Omron CX-Programmer project 新工程 (CX-Programmer 9.73)

# PLC 新PLC1: CJ1M CPU21

## Program 新程序1 (cyclic task 0)
; 这个PLC程序是我为正佳广场四楼设计的楼宇自动化控制系统。系统控制的物理设备包括照明设备、空调设备和电梯设备。系统启动时，只有在PLC上电信号为真时，照明系统电源、空调系统电源和电梯系统电源才会被激活，确保设备电源正常供应。随后，当系统启动信号为真时，系统进入运行状态，操作人员可以通过触摸屏模式选择信号选择照明模式。此时，照明控制信号置位，照明系统电源启动照明设备，为商场提供适宜的照明环境。若需调整亮度，触摸屏亮度调整信号会触发亮度调节，但这必须在系统启动信号为真的情况下才能生效，以避免未启动时误操作。通过定时器控制设备运行时间，确保设备在规定时间内完成任务。若定时器未能在预设时间内完成，系统故障指示灯会被点亮，提示操作人员检查系统状态。操作人员通过触摸屏操作信号触发系统运行输出，但系统运行输出仅在系统启动信号为真时才会被置位，防止未授权的操作影响系统。通过CMP指令比较数据寄存器的值，若检测到异常，照明故障指示灯或空调故障指示灯会被点亮，具体取决于故障来源。同时，报警灯在任何故障发生时都会点亮，向操作人员发出警示。

### Section 段1

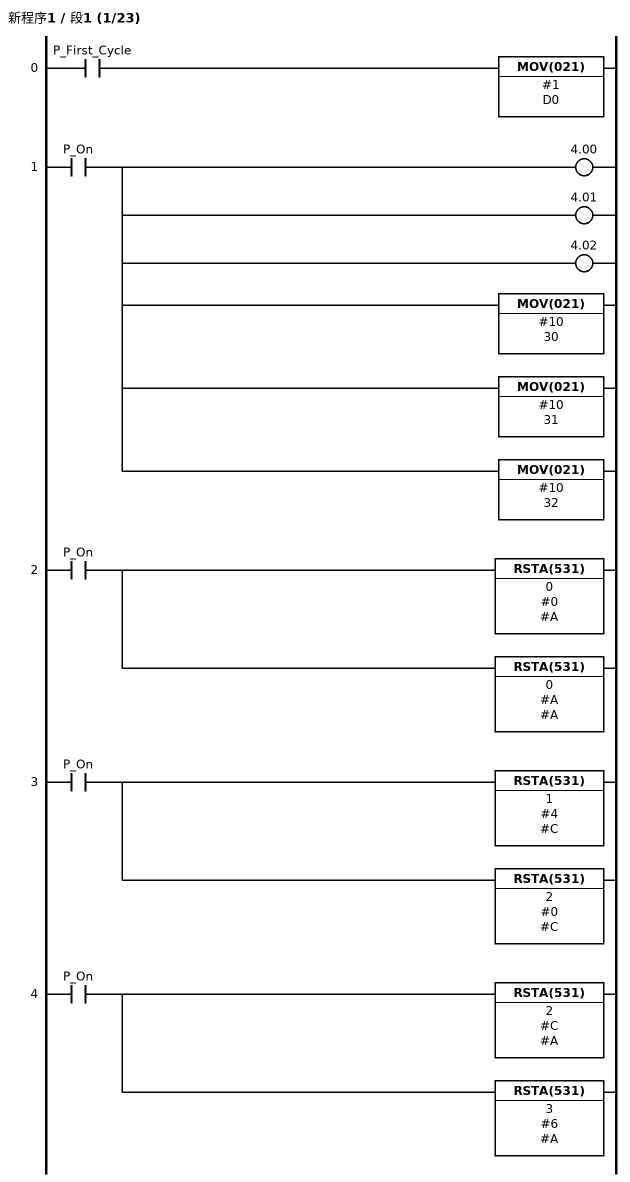
; rung 0
LD P_First_Cycle
MOV(021) #1 D0
; rung 1
LD P_On
OUT 4.00
OUT 4.01
OUT 4.02
MOV(021) #10 30
MOV(021) #10 31
MOV(021) #10 32
; rung 2
LD P_On
RSTA(531) 0 #0 #A
RSTA(531) 0 #A #A
; rung 3
LD P_On
RSTA(531) 1 #4 #C
RSTA(531) 2 #0 #C
; rung 4
LD P_On
RSTA(531) 2 #C #A
RSTA(531) 3 #6 #A

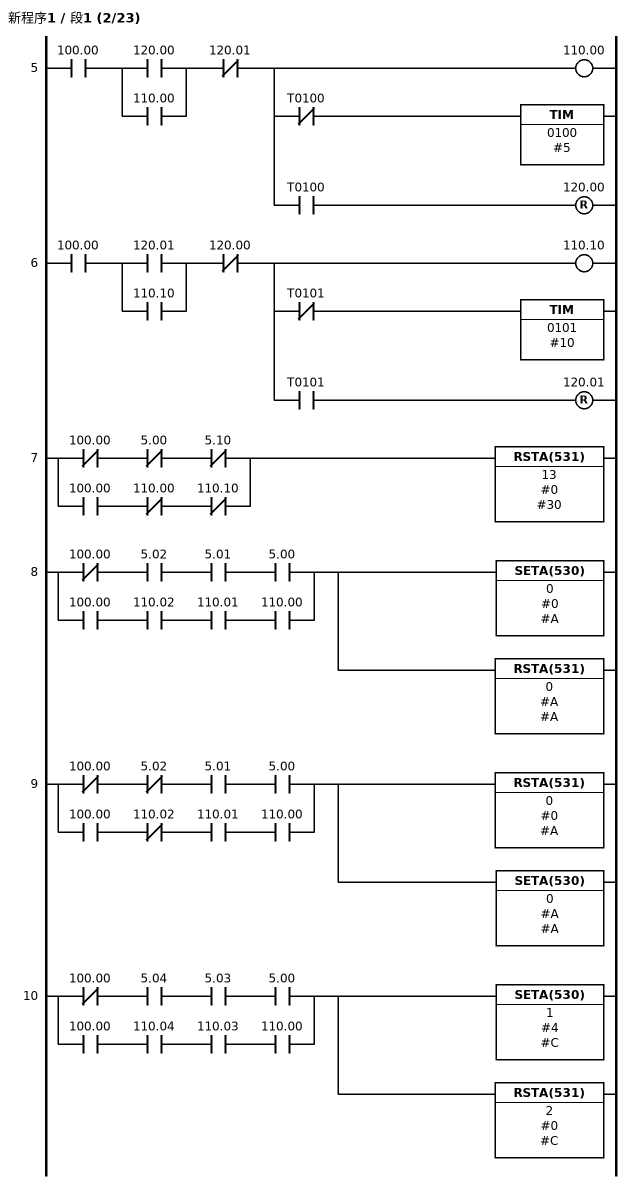
; rung 5
LD 100.00
LD 120.00
OR 110.00
ANDLD
ANDNOT 120.01
OUT TR0
OUT 110.00
ANDNOT T0100
TIM 0100 #5
LD TR0
AND T0100
RSET 120.00
; rung 6
LD 100.00
LD 120.01
OR 110.10
ANDLD
ANDNOT 120.00
OUT TR0
OUT 110.10
ANDNOT T0101
TIM 0101 #10
LD TR0
AND T0101
RSET 120.01
; rung 7
LDNOT 100.00
ANDNOT 5.00
ANDNOT 5.10
LD 100.00
ANDNOT 110.00
ANDNOT 110.10
ORLD
RSTA(531) 13 #0 #30
; rung 8
LDNOT 100.00
AND 5.02
AND 5.01
AND 5.00
LD 100.00
AND 110.02
AND 110.01
AND 110.00
ORLD
SETA(530) 0 #0 #A
RSTA(531) 0 #A #A
; rung 9
LDNOT 100.00
ANDNOT 5.02
AND 5.01
AND 5.00
LD 100.00
ANDNOT 110.02
AND 110.01
AND 110.00
ORLD
RSTA(531) 0 #0 #A
SETA(530) 0 #A #A
; rung 10
LDNOT 100.00
AND 5.04
AND 5.03
AND 5.00
LD 100.00
AND 110.04
AND 110.03
AND 110.00
ORLD
SETA(530) 1 #4 #C
RSTA(531) 2 #0 #C

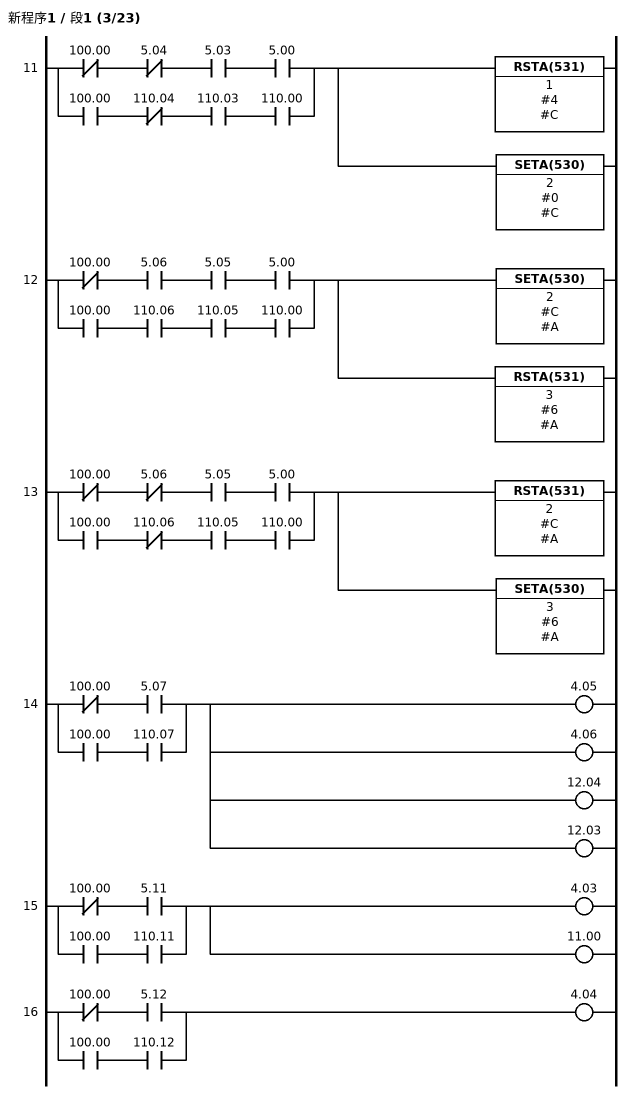
; rung 11
LDNOT 100.00
ANDNOT 5.04
AND 5.03
AND 5.00
LD 100.00
ANDNOT 110.04
AND 110.03
AND 110.00
ORLD
RSTA(531) 1 #4 #C
SETA(530) 2 #0 #C
; rung 12
LDNOT 100.00
AND 5.06
AND 5.05
AND 5.00
LD 100.00
AND 110.06
AND 110.05
AND 110.00
ORLD
SETA(530) 2 #C #A
RSTA(531) 3 #6 #A
; rung 13
LDNOT 100.00
ANDNOT 5.06
AND 5.05
AND 5.00
LD 100.00
ANDNOT 110.06
AND 110.05
AND 110.00
ORLD
RSTA(531) 2 #C #A
SETA(530) 3 #6 #A
; rung 14
LDNOT 100.00
AND 5.07
LD 100.00
AND 110.07
ORLD
OUT 4.05
OUT 4.06
OUT 12.04
OUT 12.03
; rung 15
LDNOT 100.00
AND 5.11
LD 100.00
AND 110.11
ORLD
OUT 4.03
OUT 11.00
; rung 16
LDNOT 100.00
AND 5.12
LD 100.00
AND 110.12
ORLD
OUT 4.04

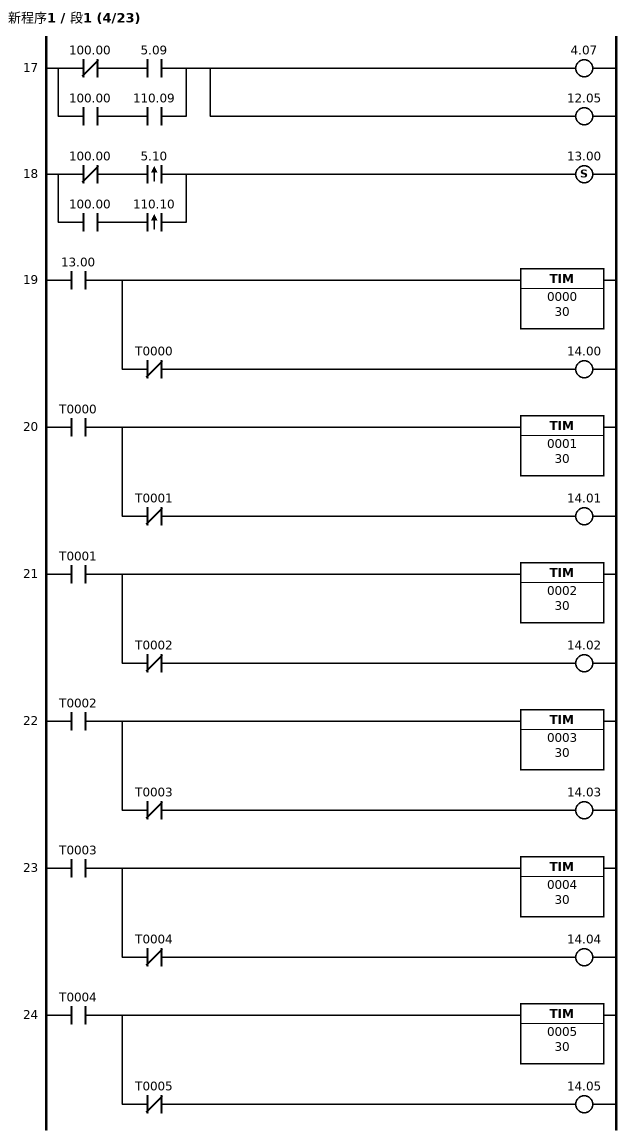
; rung 17
LDNOT 100.00
AND 5.09
LD 100.00
AND 110.09
ORLD
OUT 4.07
OUT 12.05
; rung 18
LDNOT 100.00
@AND 5.10
LD 100.00
@AND 110.10
ORLD
SET 13.00
; rung 19
LD 13.00
TIM 0000 30
ANDNOT T0000
OUT 14.00
; rung 20
LD T0000
TIM 0001 30
ANDNOT T0001
OUT 14.01
; rung 21
LD T0001
TIM 0002 30
ANDNOT T0002
OUT 14.02
; rung 22
LD T0002
TIM 0003 30
ANDNOT T0003
OUT 14.03
; rung 23
LD T0003
TIM 0004 30
ANDNOT T0004
OUT 14.04
; rung 24
LD T0004
TIM 0005 30
ANDNOT T0005
OUT 14.05

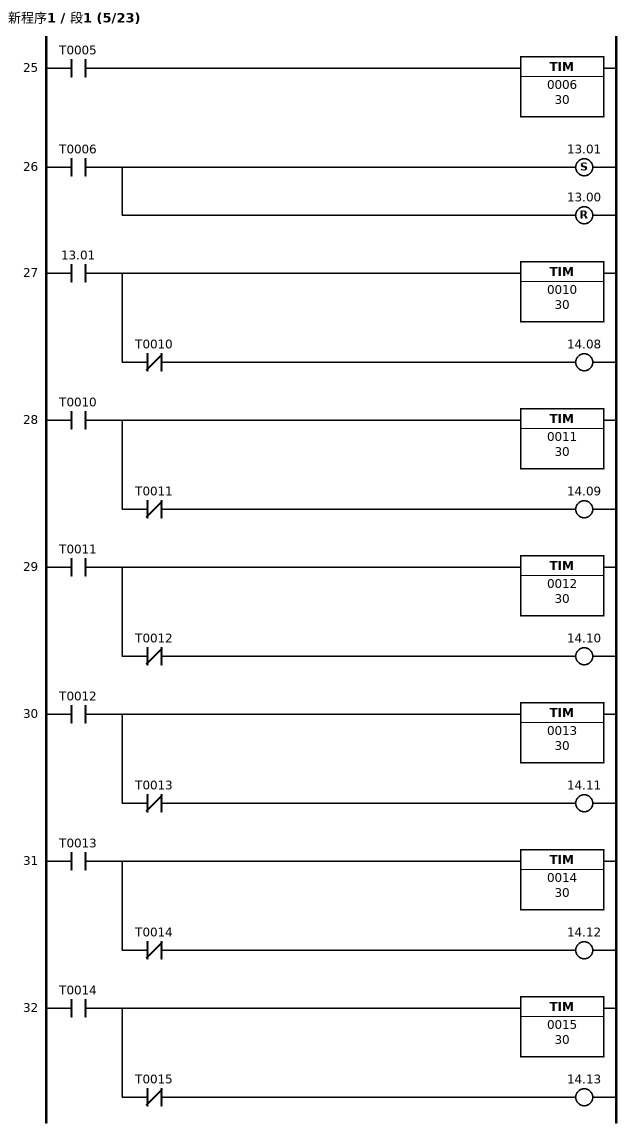
; rung 25
LD T0005
TIM 0006 30
; rung 26
LD T0006
SET 13.01
RSET 13.00
; rung 27
LD 13.01
TIM 0010 30
ANDNOT T0010
OUT 14.08
; rung 28
LD T0010
TIM 0011 30
ANDNOT T0011
OUT 14.09
; rung 29
LD T0011
TIM 0012 30
ANDNOT T0012
OUT 14.10
; rung 30
LD T0012
TIM 0013 30
ANDNOT T0013
OUT 14.11
; rung 31
LD T0013
TIM 0014 30
ANDNOT T0014
OUT 14.12
; rung 32
LD T0014
TIM 0015 30
ANDNOT T0015
OUT 14.13

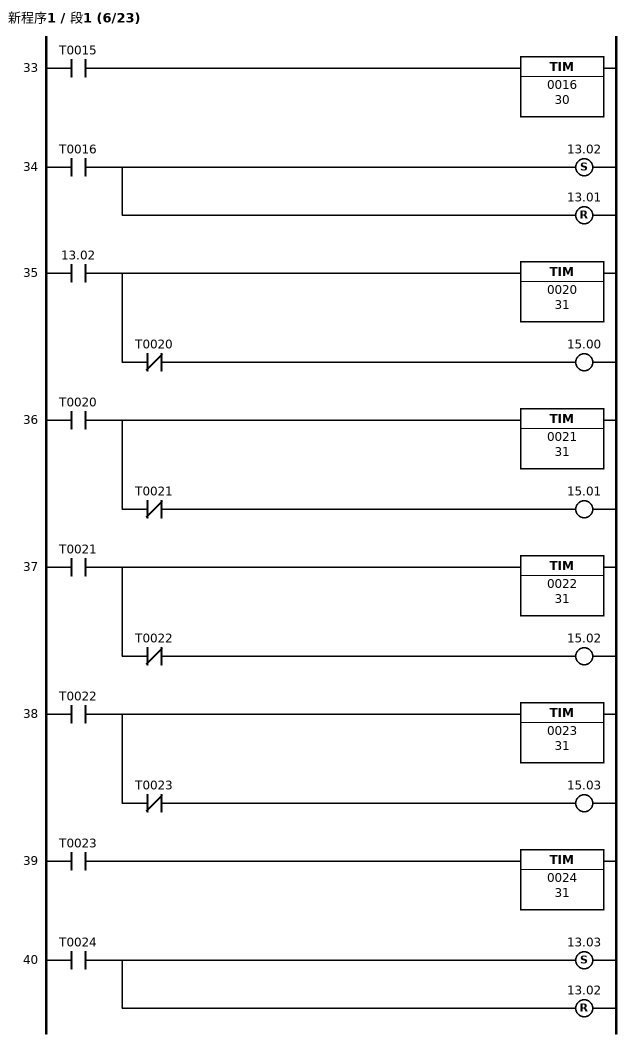
; rung 33
LD T0015
TIM 0016 30
; rung 34
LD T0016
SET 13.02
RSET 13.01
; rung 35
LD 13.02
TIM 0020 31
ANDNOT T0020
OUT 15.00
; rung 36
LD T0020
TIM 0021 31
ANDNOT T0021
OUT 15.01
; rung 37
LD T0021
TIM 0022 31
ANDNOT T0022
OUT 15.02
; rung 38
LD T0022
TIM 0023 31
ANDNOT T0023
OUT 15.03
; rung 39
LD T0023
TIM 0024 31
; rung 40
LD T0024
SET 13.03
RSET 13.02

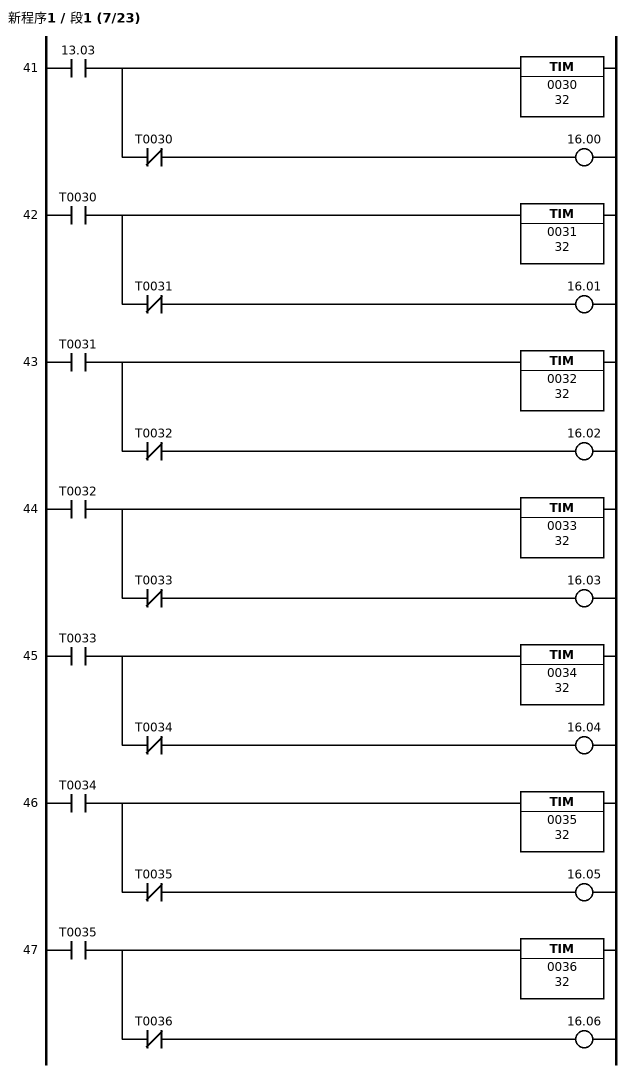
; rung 41
LD 13.03
TIM 0030 32
ANDNOT T0030
OUT 16.00
; rung 42
LD T0030
TIM 0031 32
ANDNOT T0031
OUT 16.01
; rung 43
LD T0031
TIM 0032 32
ANDNOT T0032
OUT 16.02
; rung 44
LD T0032
TIM 0033 32
ANDNOT T0033
OUT 16.03
; rung 45
LD T0033
TIM 0034 32
ANDNOT T0034
OUT 16.04
; rung 46
LD T0034
TIM 0035 32
ANDNOT T0035
OUT 16.05
; rung 47
LD T0035
TIM 0036 32
ANDNOT T0036
OUT 16.06

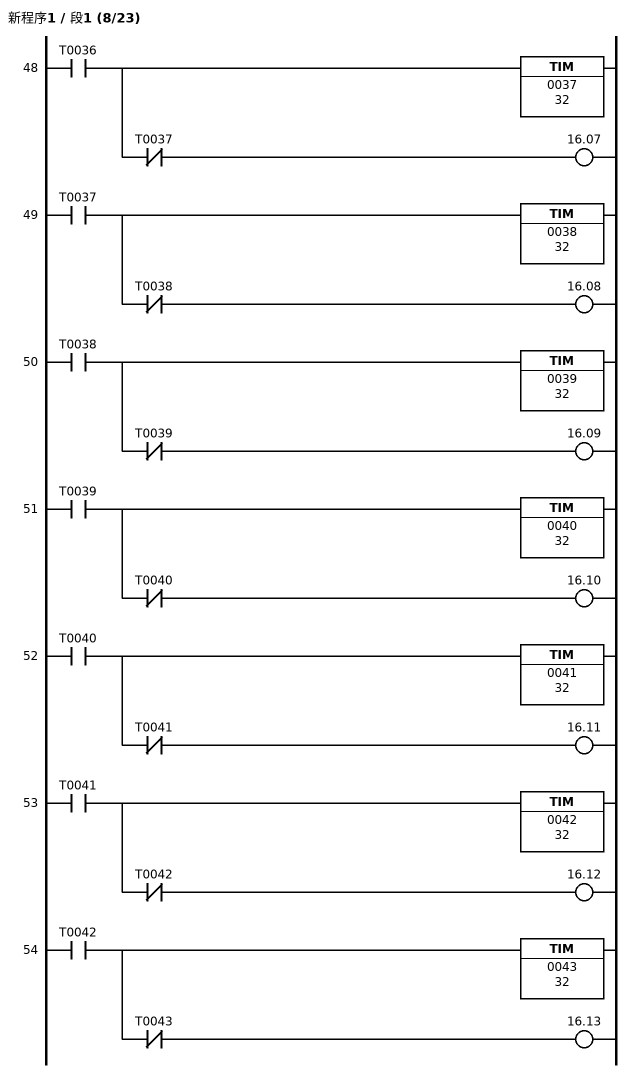
; rung 48
LD T0036
TIM 0037 32
ANDNOT T0037
OUT 16.07
; rung 49
LD T0037
TIM 0038 32
ANDNOT T0038
OUT 16.08
; rung 50
LD T0038
TIM 0039 32
ANDNOT T0039
OUT 16.09
; rung 51
LD T0039
TIM 0040 32
ANDNOT T0040
OUT 16.10
; rung 52
LD T0040
TIM 0041 32
ANDNOT T0041
OUT 16.11
; rung 53
LD T0041
TIM 0042 32
ANDNOT T0042
OUT 16.12
; rung 54
LD T0042
TIM 0043 32
ANDNOT T0043
OUT 16.13

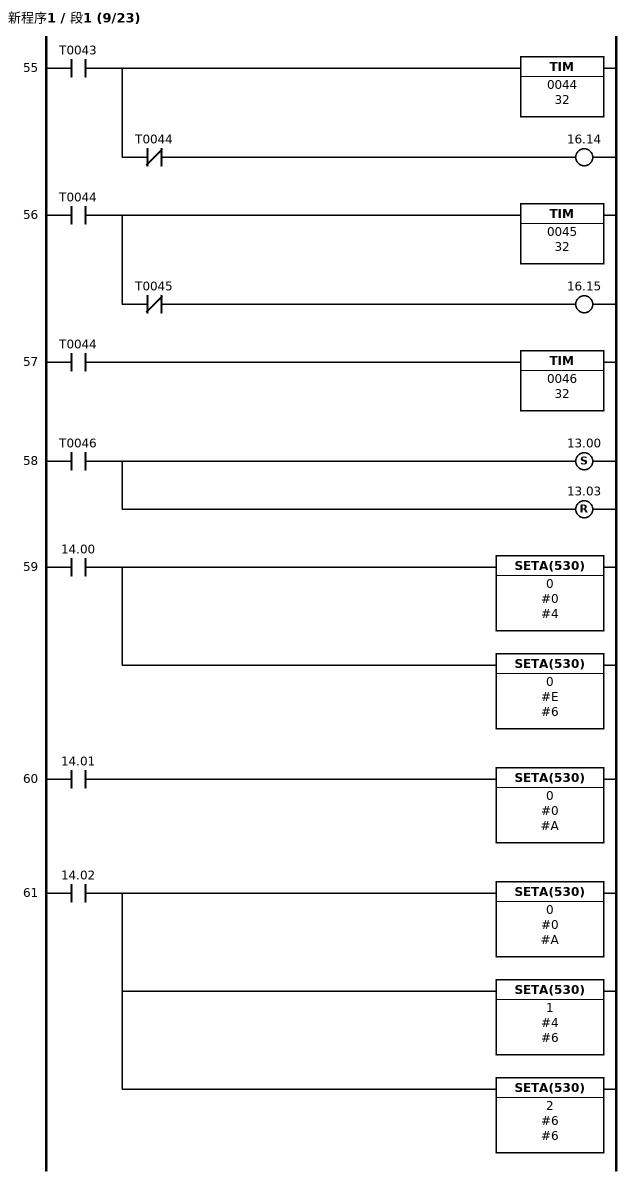
; rung 55
LD T0043
TIM 0044 32
ANDNOT T0044
OUT 16.14
; rung 56
LD T0044
TIM 0045 32
ANDNOT T0045
OUT 16.15
; rung 57
LD T0044
TIM 0046 32
; rung 58
LD T0046
SET 13.00
RSET 13.03
; rung 59
LD 14.00
SETA(530) 0 #0 #4
SETA(530) 0 #E #6
; rung 60
LD 14.01
SETA(530) 0 #0 #A
; rung 61
LD 14.02
SETA(530) 0 #0 #A
SETA(530) 1 #4 #6
SETA(530) 2 #6 #6

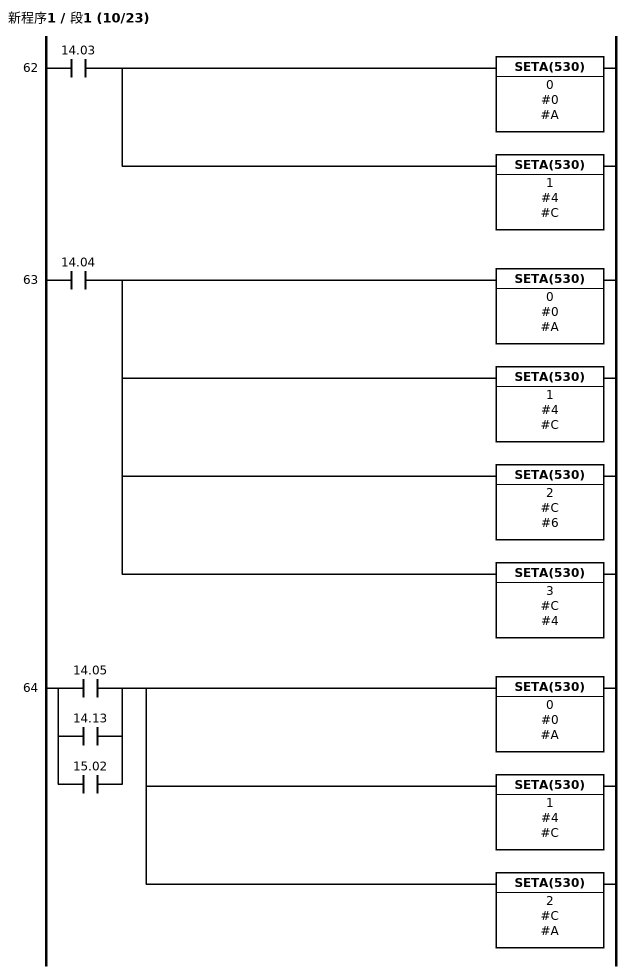
; rung 62
LD 14.03
SETA(530) 0 #0 #A
SETA(530) 1 #4 #C
; rung 63
LD 14.04
SETA(530) 0 #0 #A
SETA(530) 1 #4 #C
SETA(530) 2 #C #6
SETA(530) 3 #C #4
; rung 64
LD 14.05
OR 14.13
OR 15.02
SETA(530) 0 #0 #A
SETA(530) 1 #4 #C
SETA(530) 2 #C #A

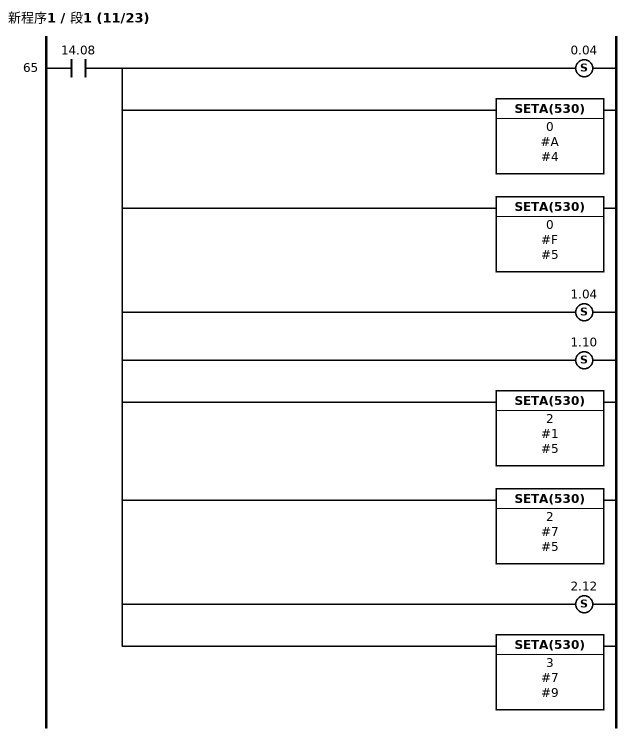
; rung 65
LD 14.08
SET 0.04
SETA(530) 0 #A #4
SETA(530) 0 #F #5
SET 1.04
SET 1.10
SETA(530) 2 #1 #5
SETA(530) 2 #7 #5
SET 2.12
SETA(530) 3 #7 #9

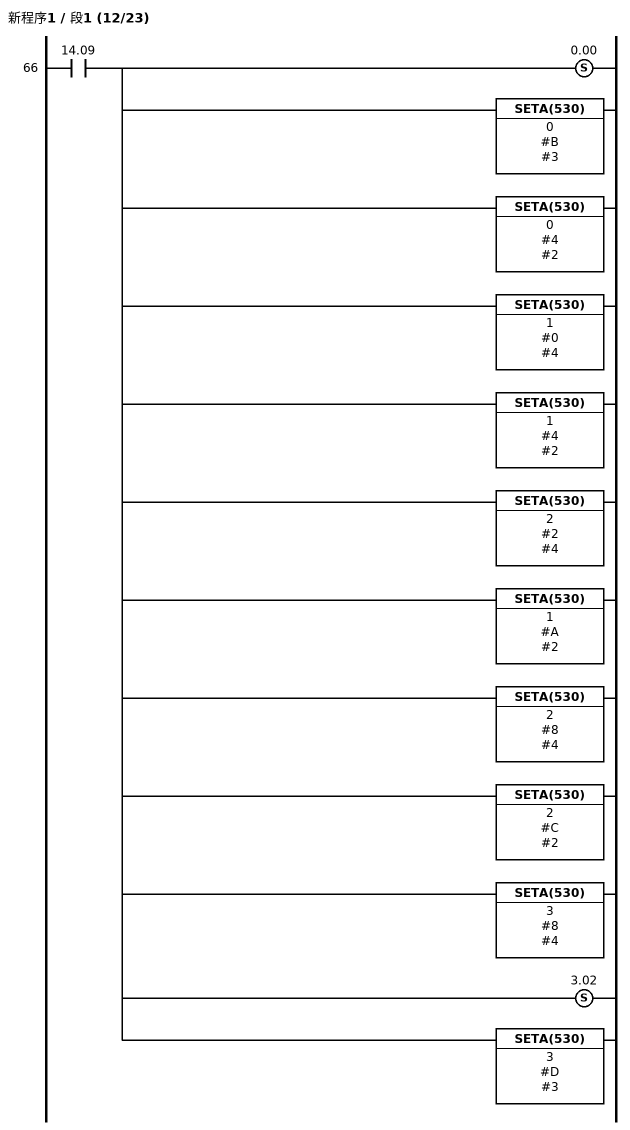
; rung 66
LD 14.09
SET 0.00
SETA(530) 0 #B #3
SETA(530) 0 #4 #2
SETA(530) 1 #0 #4
SETA(530) 1 #4 #2
SETA(530) 2 #2 #4
SETA(530) 1 #A #2
SETA(530) 2 #8 #4
SETA(530) 2 #C #2
SETA(530) 3 #8 #4
SET 3.02
SETA(530) 3 #D #3

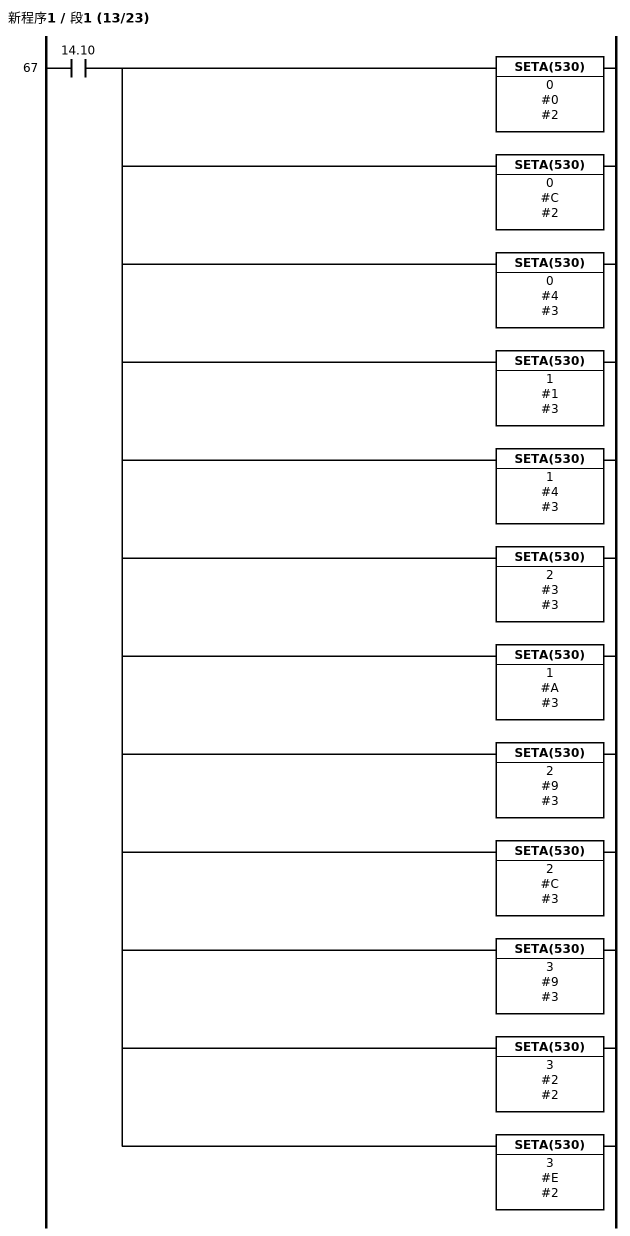
; rung 67
LD 14.10
SETA(530) 0 #0 #2
SETA(530) 0 #C #2
SETA(530) 0 #4 #3
SETA(530) 1 #1 #3
SETA(530) 1 #4 #3
SETA(530) 2 #3 #3
SETA(530) 1 #A #3
SETA(530) 2 #9 #3
SETA(530) 2 #C #3
SETA(530) 3 #9 #3
SETA(530) 3 #2 #2
SETA(530) 3 #E #2

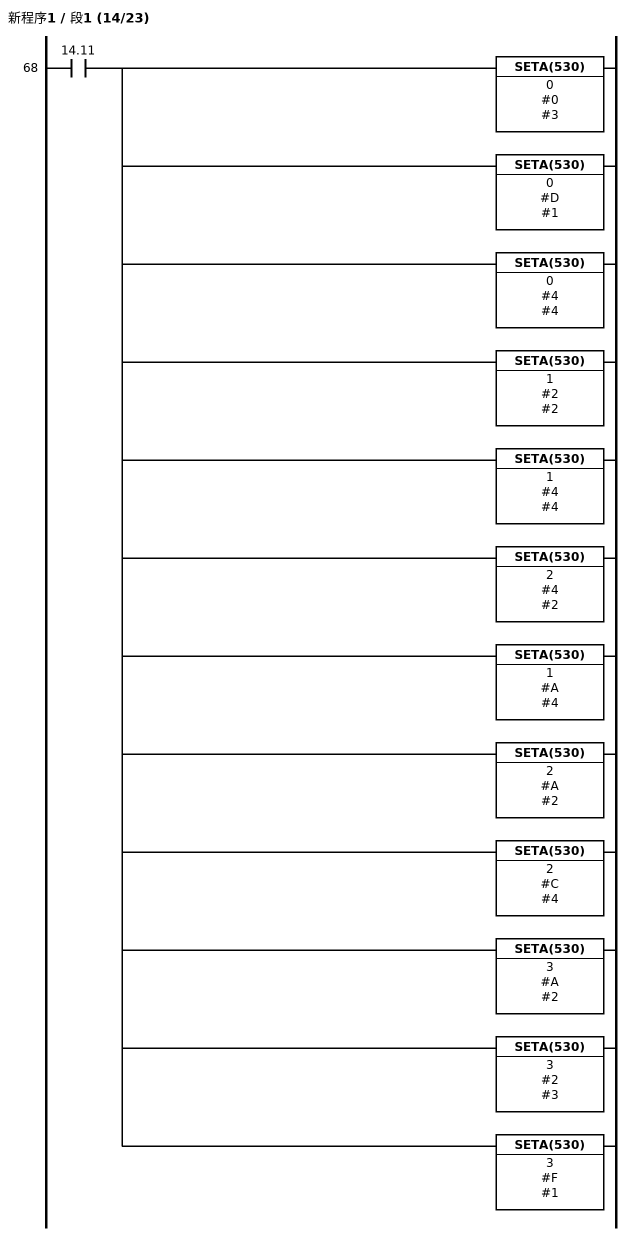
; rung 68
LD 14.11
SETA(530) 0 #0 #3
SETA(530) 0 #D #1
SETA(530) 0 #4 #4
SETA(530) 1 #2 #2
SETA(530) 1 #4 #4
SETA(530) 2 #4 #2
SETA(530) 1 #A #4
SETA(530) 2 #A #2
SETA(530) 2 #C #4
SETA(530) 3 #A #2
SETA(530) 3 #2 #3
SETA(530) 3 #F #1

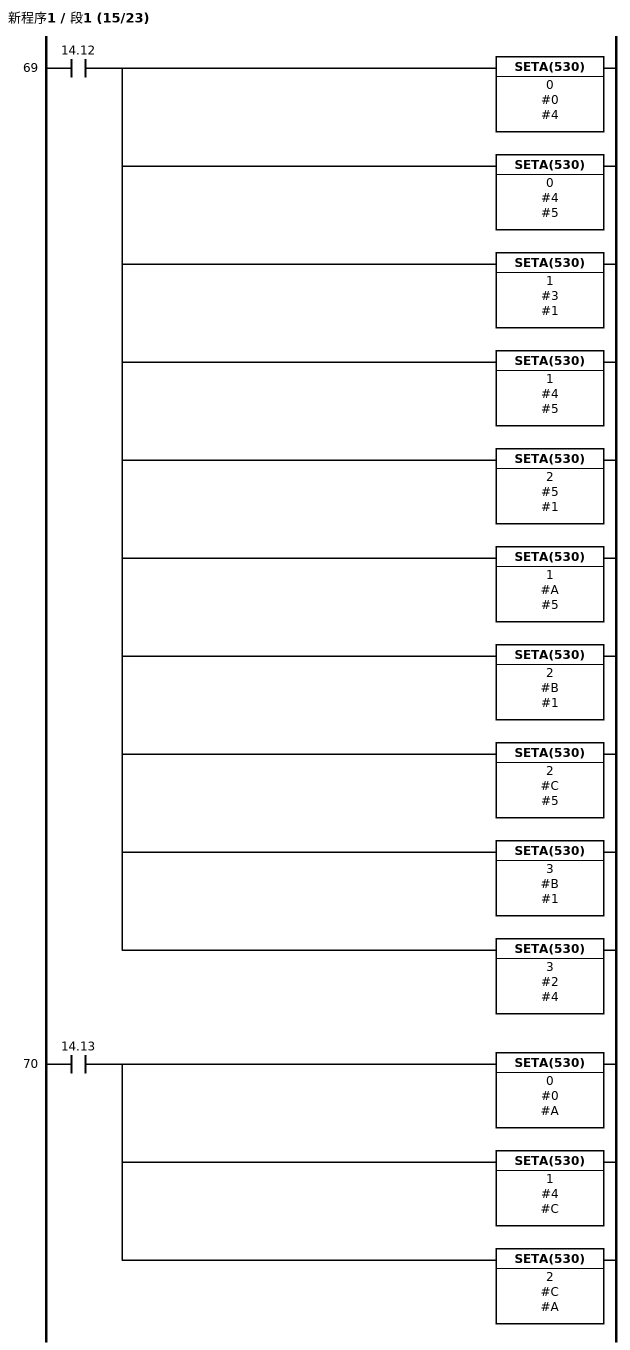
; rung 69
LD 14.12
SETA(530) 0 #0 #4
SETA(530) 0 #4 #5
SETA(530) 1 #3 #1
SETA(530) 1 #4 #5
SETA(530) 2 #5 #1
SETA(530) 1 #A #5
SETA(530) 2 #B #1
SETA(530) 2 #C #5
SETA(530) 3 #B #1
SETA(530) 3 #2 #4
; rung 70
LD 14.13
SETA(530) 0 #0 #A
SETA(530) 1 #4 #C
SETA(530) 2 #C #A

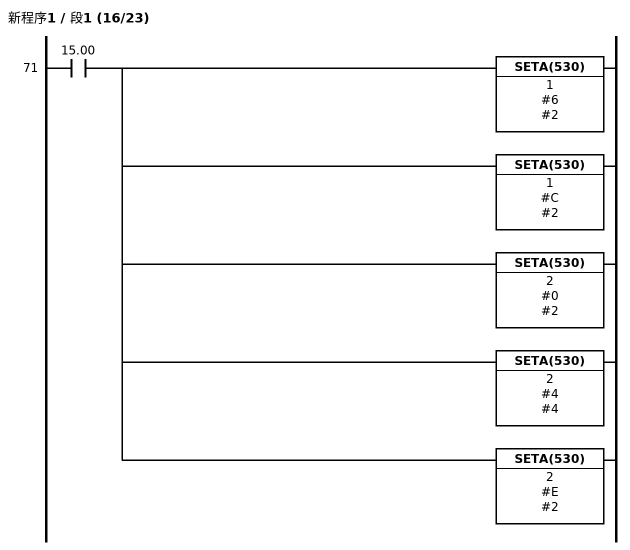
; rung 71
LD 15.00
SETA(530) 1 #6 #2
SETA(530) 1 #C #2
SETA(530) 2 #0 #2
SETA(530) 2 #4 #4
SETA(530) 2 #E #2

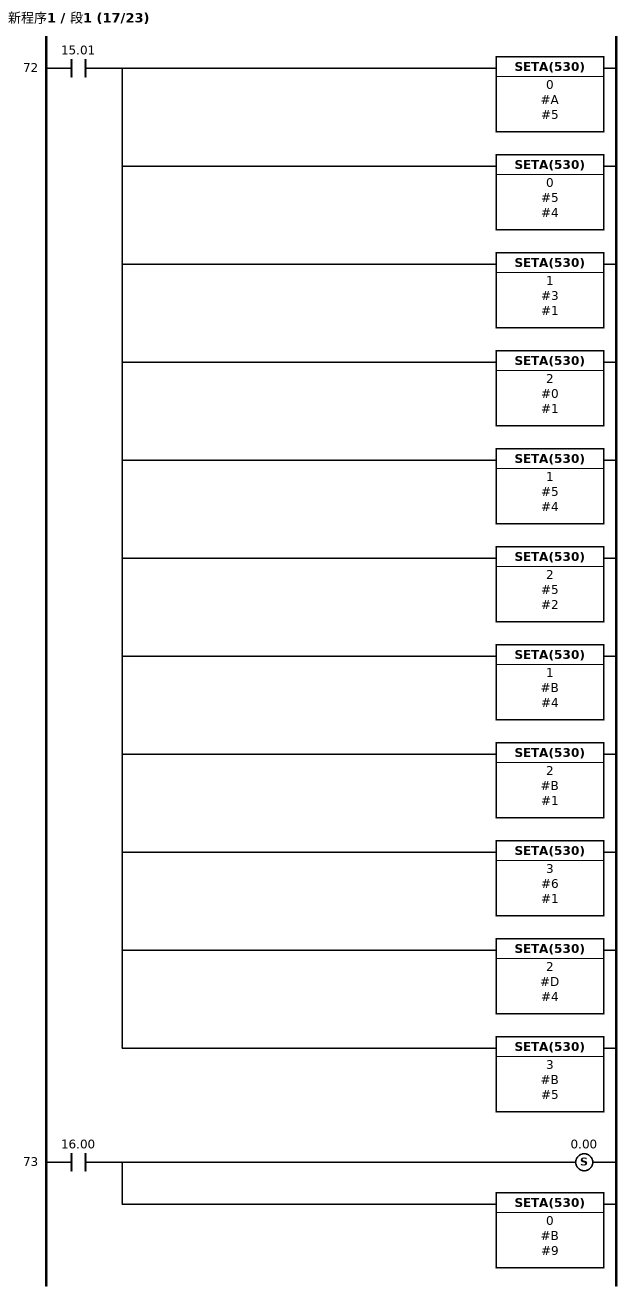
; rung 72
LD 15.01
SETA(530) 0 #A #5
SETA(530) 0 #5 #4
SETA(530) 1 #3 #1
SETA(530) 2 #0 #1
SETA(530) 1 #5 #4
SETA(530) 2 #5 #2
SETA(530) 1 #B #4
SETA(530) 2 #B #1
SETA(530) 3 #6 #1
SETA(530) 2 #D #4
SETA(530) 3 #B #5
; rung 73
LD 16.00
SET 0.00
SETA(530) 0 #B #9

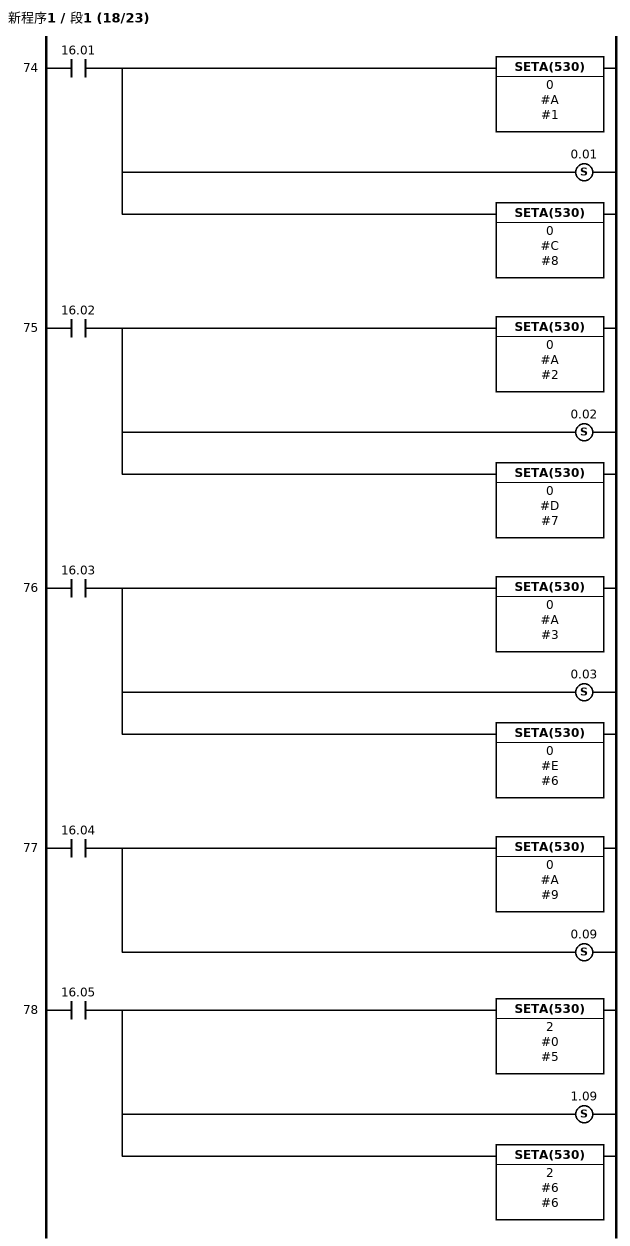
; rung 74
LD 16.01
SETA(530) 0 #A #1
SET 0.01
SETA(530) 0 #C #8
; rung 75
LD 16.02
SETA(530) 0 #A #2
SET 0.02
SETA(530) 0 #D #7
; rung 76
LD 16.03
SETA(530) 0 #A #3
SET 0.03
SETA(530) 0 #E #6
; rung 77
LD 16.04
SETA(530) 0 #A #9
SET 0.09
; rung 78
LD 16.05
SETA(530) 2 #0 #5
SET 1.09
SETA(530) 2 #6 #6

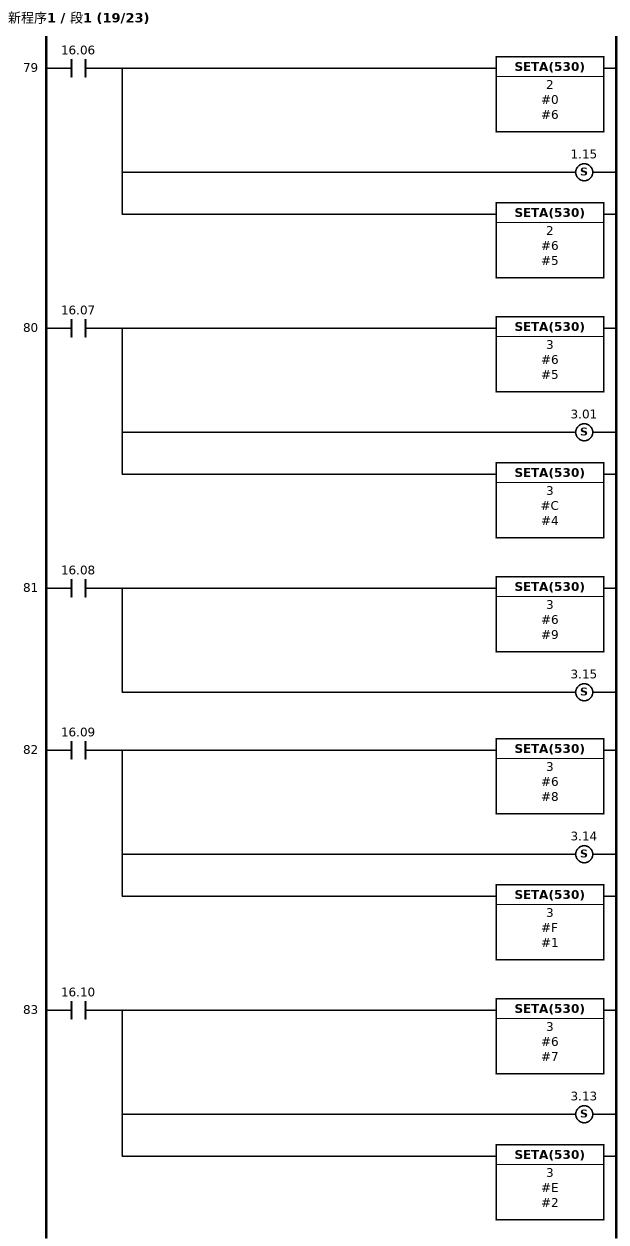
; rung 79
LD 16.06
SETA(530) 2 #0 #6
SET 1.15
SETA(530) 2 #6 #5
; rung 80
LD 16.07
SETA(530) 3 #6 #5
SET 3.01
SETA(530) 3 #C #4
; rung 81
LD 16.08
SETA(530) 3 #6 #9
SET 3.15
; rung 82
LD 16.09
SETA(530) 3 #6 #8
SET 3.14
SETA(530) 3 #F #1
; rung 83
LD 16.10
SETA(530) 3 #6 #7
SET 3.13
SETA(530) 3 #E #2

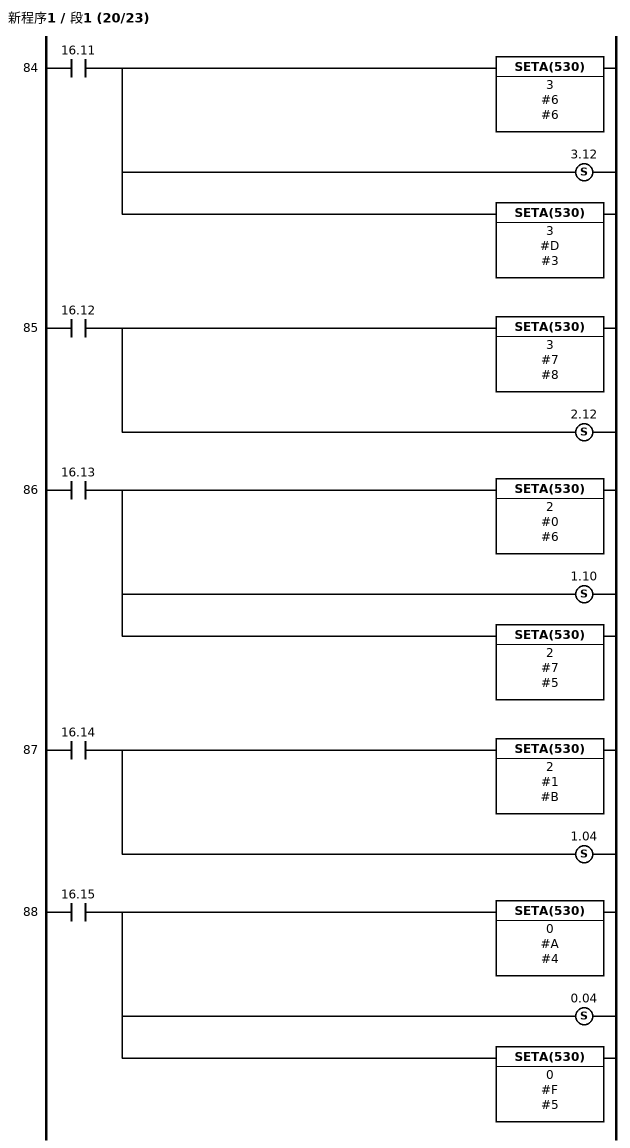
; rung 84
LD 16.11
SETA(530) 3 #6 #6
SET 3.12
SETA(530) 3 #D #3
; rung 85
LD 16.12
SETA(530) 3 #7 #8
SET 2.12
; rung 86
LD 16.13
SETA(530) 2 #0 #6
SET 1.10
SETA(530) 2 #7 #5
; rung 87
LD 16.14
SETA(530) 2 #1 #B
SET 1.04
; rung 88
LD 16.15
SETA(530) 0 #A #4
SET 0.04
SETA(530) 0 #F #5

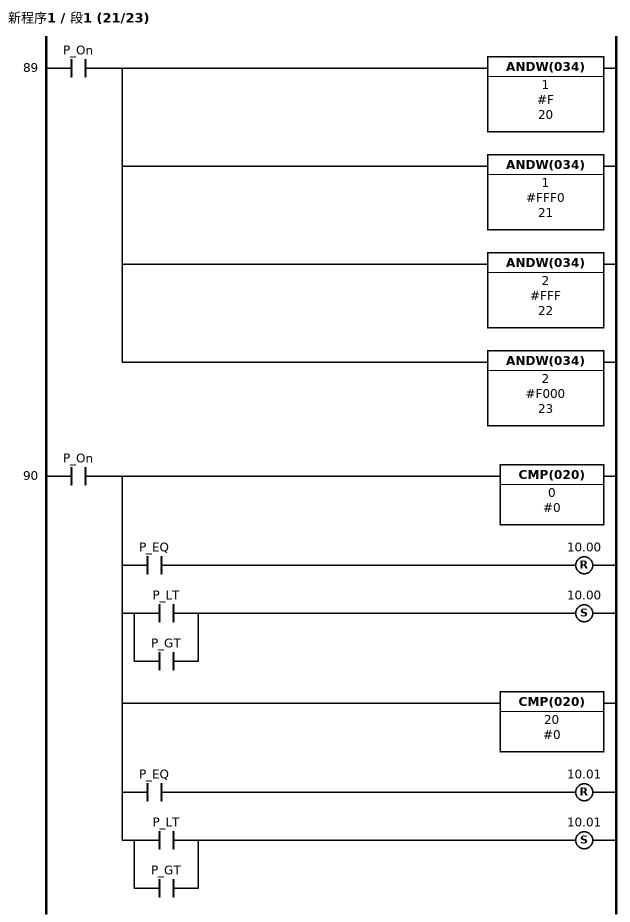
; rung 89
LD P_On
ANDW(034) 1 #F 20
ANDW(034) 1 #FFF0 21
ANDW(034) 2 #FFF 22
ANDW(034) 2 #F000 23
; rung 90
LD P_On
OUT TR0
CMP(020) 0 #0
AND P_EQ
RSET 10.00
LD TR0
LD P_LT
OR P_GT
ANDLD
SET 10.00
LD TR0
CMP(020) 20 #0
AND P_EQ
RSET 10.01
LD TR0
LD P_LT
OR P_GT
ANDLD
SET 10.01

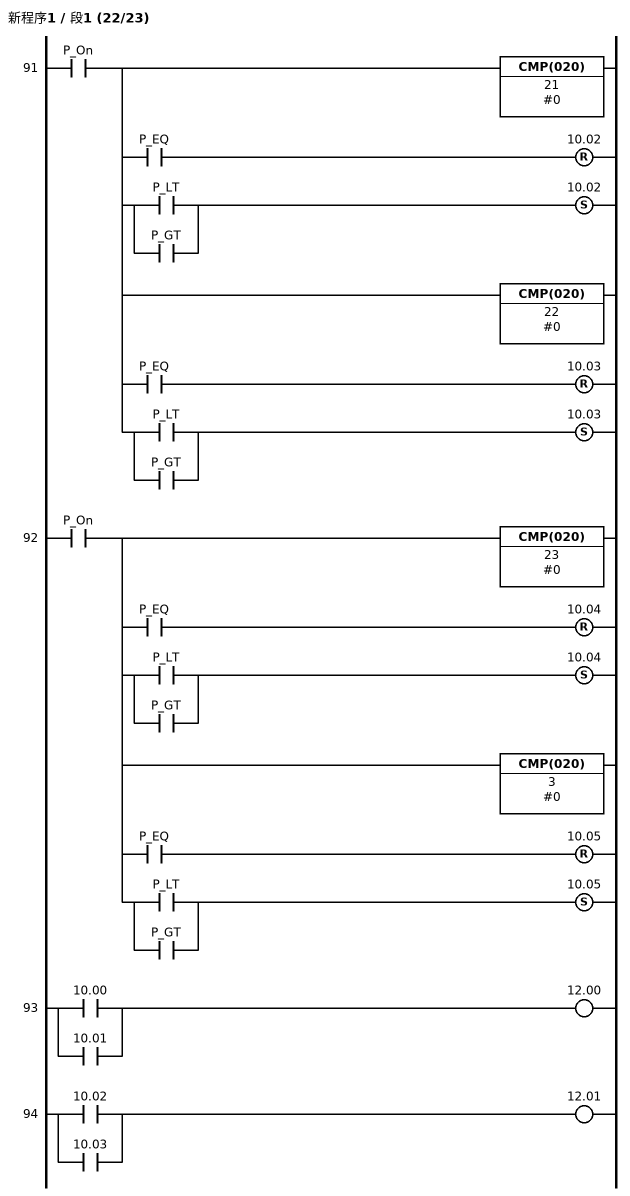
; rung 91
LD P_On
OUT TR0
CMP(020) 21 #0
AND P_EQ
RSET 10.02
LD TR0
LD P_LT
OR P_GT
ANDLD
SET 10.02
LD TR0
CMP(020) 22 #0
AND P_EQ
RSET 10.03
LD TR0
LD P_LT
OR P_GT
ANDLD
SET 10.03
; rung 92
LD P_On
OUT TR0
CMP(020) 23 #0
AND P_EQ
RSET 10.04
LD TR0
LD P_LT
OR P_GT
ANDLD
SET 10.04
LD TR0
CMP(020) 3 #0
AND P_EQ
RSET 10.05
LD TR0
LD P_LT
OR P_GT
ANDLD
SET 10.05
; rung 93
LD 10.00
OR 10.01
OUT 12.00
; rung 94
LD 10.02
OR 10.03
OUT 12.01

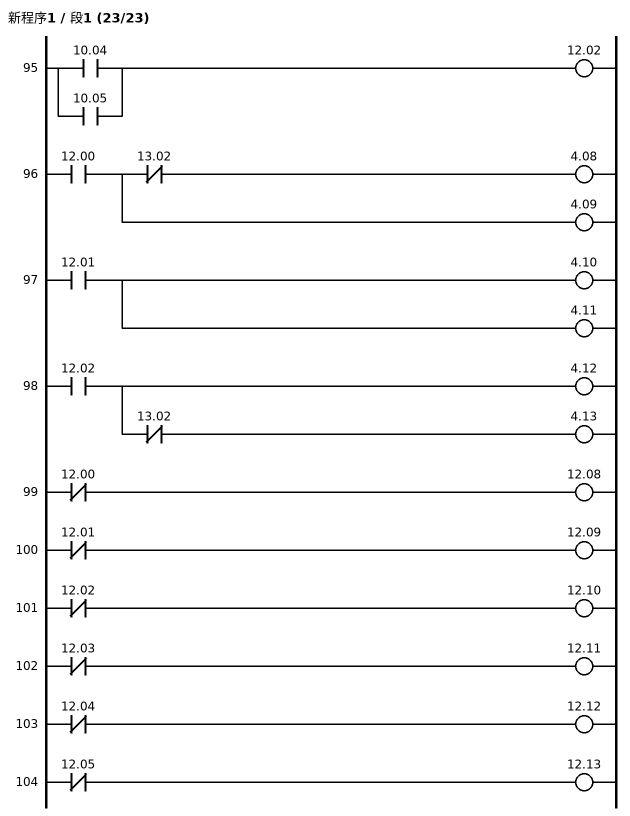
; rung 95
LD 10.04
OR 10.05
OUT 12.02
; rung 96
LD 12.00
OUT TR0
ANDNOT 13.02
OUT 4.08
LD TR0
OUT 4.09
; rung 97
LD 12.01
OUT 4.10
OUT 4.11
; rung 98
LD 12.02
OUT 4.12
ANDNOT 13.02
OUT 4.13
; rung 99
LDNOT 12.00
OUT 12.08
; rung 100
LDNOT 12.01
OUT 12.09
; rung 101
LDNOT 12.02
OUT 12.10
; rung 102
LDNOT 12.03
OUT 12.11
; rung 103
LDNOT 12.04
OUT 12.12
; rung 104
LDNOT 12.05
OUT 12.13
; rung 105
END(001)

### Section 段2
; rung 0
END(001)